TEXTLIST MTCSConfigTabsTextList
  0 = 'Instruments'
   = ''
END_TEXTLIST

(* stored: Version 1.1.0.1, ProductVersion 3.1.4018.5
   TextList MTCSConfigTabsTextList: Id {8eb9fc50-b5aa-447f-961a-f392d7911d94} *)
